FUNCTION_BLOCK ControlLogic (* Composite Function Block Type *)
  (* Standard: 61499-2 *)
  (* Version 0.0, 5/26/2025, Guillaume De Martino, Schneider Electric, template *)
  PACKAGE Main;
  (* 1 - FUNCTIONAL PARENT INTERFACE *)
  (* 2 - FUNCTIONAL SIBLINGS INTERFACE *)
  (* 5 - LOGICS *)
  (* 6 - HMI INTERFACE *)
  (* 5.A - FUNCTIONAL BEHAVIOR *)
  (* 5.E - STATIC PARAMETERS MANAGEMENT *)
  (* IN-DATA ELABORATION *)
  (* OUT-DATA ELABORATION *)
END_FUNCTION_BLOCK
